// TIA Portal V17 export
// export: Created 2025-03-07T09:16:41.622432Z, ExportSetting WithDefaults, DisplayName Totally Integrated Automation Portal, DisplayVersion V17 Update 8, DisplayName TIA Portal Openness, DisplayVersion V17 Update 8, DisplayName TIA Portal Version Control Interface, DisplayVersion V17, DisplayName SINAMICS Startdrive Advanced, DisplayVersion V17 SP2, DisplayName SINAMICS Startdrive G110M, G120, G120C, G120D, G120P, G115D, DisplayVersion V17 SP2, DisplayName SINAMICS Startdrive G130, G150, S120, S150, SINAMICS MV, S210, DisplayVersion V17 SP2, DisplayName STEP 7 Professional, DisplayVersion V17 Update 8, DisplayName SINUMERIK ONE STEP 7 Toolbox, DisplayVersion V17 Update 12, DisplayName SINUMERIK 840D sl STEP 7 Toolbox, DisplayVersion V17 Update 12, DisplayName STEP 7 Safety, DisplayVersion V17 Update 6, DisplayName WinCC Advanced, DisplayVersion V17 Update 8
FUNCTION "FC2441_MACHINE_STATUS" : Void   // FC2441, LAD
{ S7_Optimized_Access := 'TRUE' }
VERSION : 0.1
// stored: AutoNumber false, IsIECCheckEnabled false, SetENOAutomatically false, UDAEnableTagReadback false
BEGIN

REGION Network 1: UNIT 01 STATION 3 CLADDING IN PROCESS
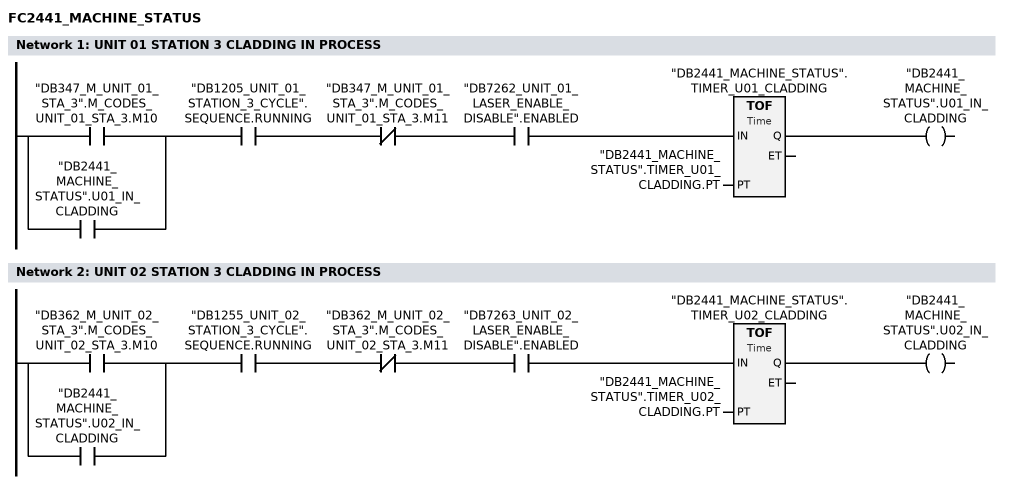
   RUNG wire#powerrail
      Contact( "DB347_M_UNIT_01_STA_3".M_CODES_UNIT_01_STA_3.M10 )
      wire#w1
      Contact( "DB1205_UNIT_01_STATION_3_CYCLE".SEQUENCE.RUNNING )
      I_Contact( "DB347_M_UNIT_01_STA_3".M_CODES_UNIT_01_STA_3.M11 )
      Contact( "DB7262_UNIT_01_LASER_ENABLE_DISABLE".ENABLED )
      { S7_Templates := "time_type := Time" } "DB2441_MACHINE_STATUS".TIMER_U01_CLADDING.TOF(pt := "DB2441_MACHINE_STATUS".TIMER_U01_CLADDING.PT, et =>)
      Coil( "DB2441_MACHINE_STATUS".U01_IN_CLADDING )
   END_RUNG
   RUNG wire#powerrail
      Contact( "DB2441_MACHINE_STATUS".U01_IN_CLADDING )
   END_RUNG wire#w1
   // the same network as SCL:
   "DB2441_MACHINE_STATUS".TIMER_U01_CLADDING.TOF(IN := ("DB347_M_UNIT_01_STA_3".M_CODES_UNIT_01_STA_3.M10 OR "DB2441_MACHINE_STATUS".U01_IN_CLADDING) AND "DB1205_UNIT_01_STATION_3_CYCLE".SEQUENCE.RUNNING AND NOT "DB347_M_UNIT_01_STA_3".M_CODES_UNIT_01_STA_3.M11 AND "DB7262_UNIT_01_LASER_ENABLE_DISABLE".ENABLED,
                           PT := "DB2441_MACHINE_STATUS".TIMER_U01_CLADDING.PT);
   "DB2441_MACHINE_STATUS".U01_IN_CLADDING := "DB2441_MACHINE_STATUS".TIMER_U01_CLADDING.Q;
END_REGION

REGION Network 2: UNIT 02 STATION 3 CLADDING IN PROCESS
   RUNG wire#powerrail
      Contact( "DB362_M_UNIT_02_STA_3".M_CODES_UNIT_02_STA_3.M10 )
      wire#w1
      Contact( "DB1255_UNIT_02_STATION_3_CYCLE".SEQUENCE.RUNNING )
      I_Contact( "DB362_M_UNIT_02_STA_3".M_CODES_UNIT_02_STA_3.M11 )
      Contact( "DB7263_UNIT_02_LASER_ENABLE_DISABLE".ENABLED )
      { S7_Templates := "time_type := Time" } "DB2441_MACHINE_STATUS".TIMER_U02_CLADDING.TOF(pt := "DB2441_MACHINE_STATUS".TIMER_U02_CLADDING.PT, et =>)
      Coil( "DB2441_MACHINE_STATUS".U02_IN_CLADDING )
   END_RUNG
   RUNG wire#powerrail
      Contact( "DB2441_MACHINE_STATUS".U02_IN_CLADDING )
   END_RUNG wire#w1
   // the same network as SCL:
   "DB2441_MACHINE_STATUS".TIMER_U02_CLADDING.TOF(IN := ("DB362_M_UNIT_02_STA_3".M_CODES_UNIT_02_STA_3.M10 OR "DB2441_MACHINE_STATUS".U02_IN_CLADDING) AND "DB1255_UNIT_02_STATION_3_CYCLE".SEQUENCE.RUNNING AND NOT "DB362_M_UNIT_02_STA_3".M_CODES_UNIT_02_STA_3.M11 AND "DB7263_UNIT_02_LASER_ENABLE_DISABLE".ENABLED,
                           PT := "DB2441_MACHINE_STATUS".TIMER_U02_CLADDING.PT);
   "DB2441_MACHINE_STATUS".U02_IN_CLADDING := "DB2441_MACHINE_STATUS".TIMER_U02_CLADDING.Q;
END_REGION
END_FUNCTION
